(* IEC 61131-3 sources: openplc_school_01/practice04/build/OpenPLC Runtime v3/src, 1 file *)

(* ---- program.st ---- *)
PROGRAM main
  VAR_INPUT
    X0 : BOOL;
    X1 : BOOL;
  END_VAR
  VAR_OUTPUT
    Y0 : BOOL;
  END_VAR

  Y0 := NOT(X1) AND NOT(X0);
END_PROGRAM

CONFIGURATION Config0

  RESOURCE Res0 ON PLC
    TASK task0(INTERVAL := T#20ms,PRIORITY := 1);
    PROGRAM instance0 WITH task0 : main;
  END_RESOURCE
END_CONFIGURATION

(*DBG:char md5[] = "5c376f10d533214feb88b87bce6b503e";*)
(*DBG:/**)
(*DBG: * This file is part of OpenPLC Runtime*)
(*DBG: **)
(*DBG: * Copyright (C) 2023 Autonomy, GP Orcullo*)
(*DBG: * Based on the work by GP Orcullo on Beremiz for uC*)
(*DBG: **)
(*DBG: * This program is free software; you can redistribute it and/or*)
(*DBG: * modify it under the terms of the GNU General Public License*)
(*DBG: * as published by the Free Software Foundation; either version 2*)
(*DBG: * of the License, or (at your option) any later version.*)
(*DBG: **)
(*DBG: * This program is distributed in the hope that it will be useful,*)
(*DBG: * but WITHOUT ANY WARRANTY; without even the implied warranty of*)
(*DBG: * MERCHANTABILITY or FITNESS FOR A PARTICULAR PURPOSE.  See the*)
(*DBG: * GNU General Public License for more details.*)
(*DBG: **)
(*DBG: * You should have received a copy of the GNU General Public License*)
(*DBG: * along with this program; If not, see <http://www.gnu.org/licenses/>.*)
(*DBG: **)
(*DBG: */*)
(*DBG:*)
(*DBG:#include <stdbool.h>*)
(*DBG:*)
(*DBG:#include "iec_types_all.h"*)
(*DBG:#include "POUS.h"*)
(*DBG:*)
(*DBG:#define SAME_ENDIANNESS      0*)
(*DBG:#define REVERSE_ENDIANNESS   1*)
(*DBG:*)
(*DBG:char plc_program_md5[] = "5c376f10d533214feb88b87bce6b503e";*)
(*DBG:*)
(*DBG:uint8_t endianness;*)
(*DBG:*)
(*DBG:*)
(*DBG:extern MAIN RES0__INSTANCE0;*)
(*DBG:*)
(*DBG:static const struct {*)
(*DBG:    void *ptr;*)
(*DBG:    __IEC_types_enum type;*)
(*DBG:} debug_vars[] = {*)
(*DBG:    {&(RES0__INSTANCE0.X0), BOOL_ENUM},*)
(*DBG:    {&(RES0__INSTANCE0.X1), BOOL_ENUM},*)
(*DBG:    {&(RES0__INSTANCE0.Y0), BOOL_ENUM},*)
(*DBG:};*)
(*DBG:*)
(*DBG:#define VAR_COUNT               3*)
(*DBG:*)
(*DBG:uint16_t get_var_count(void)*)
(*DBG:{*)
(*DBG:    return VAR_COUNT;*)
(*DBG:}*)
(*DBG:*)
(*DBG:size_t get_var_size(size_t idx)*)
(*DBG:{*)
(*DBG:    if (idx >= VAR_COUNT)*)
(*DBG:    {*)
(*DBG:        return 0;*)
(*DBG:    }*)
(*DBG:    switch (debug_vars[idx].type) {*)
(*DBG:    case BOOL_ENUM:*)
(*DBG:        return sizeof(BOOL);*)
(*DBG:    default:*)
(*DBG:        return 0;*)
(*DBG:    }*)
(*DBG:}*)
(*DBG:*)
(*DBG:void *get_var_addr(size_t idx)*)
(*DBG:{*)
(*DBG:    void *ptr = debug_vars[idx].ptr;*)
(*DBG:*)
(*DBG:    switch (debug_vars[idx].type) {*)
(*DBG:    case BOOL_ENUM:*)
(*DBG:        return (void *)&((__IEC_BOOL_t *) ptr)->value;*)
(*DBG:    default:*)
(*DBG:        return 0;*)
(*DBG:    }*)
(*DBG:}*)
(*DBG:*)
(*DBG:void force_var(size_t idx, bool forced, void *val)*)
(*DBG:{*)
(*DBG:    void *ptr = debug_vars[idx].ptr;*)
(*DBG:*)
(*DBG:    if (forced) {*)
(*DBG:        size_t var_size = get_var_size(idx);*)
(*DBG:        switch (debug_vars[idx].type) {*)
(*DBG:        case BOOL_ENUM: {*)
(*DBG:            memcpy(&((__IEC_BOOL_t *) ptr)->value, val, var_size);*)
(*DBG:            ((__IEC_BOOL_t *) ptr)->flags |= __IEC_FORCE_FLAG;*)
(*DBG:            break;*)
(*DBG:        }*)
(*DBG:    *)
(*DBG:        default:*)
(*DBG:            break;*)
(*DBG:        }*)
(*DBG:    } else {*)
(*DBG:        switch (debug_vars[idx].type) {*)
(*DBG:        case BOOL_ENUM:*)
(*DBG:            ((__IEC_BOOL_t *) ptr)->flags &= ~__IEC_FORCE_FLAG;*)
(*DBG:            break;*)
(*DBG:        default:*)
(*DBG:            break;*)
(*DBG:        }*)
(*DBG:    }*)
(*DBG:}*)
(*DBG:*)
(*DBG:void swap_bytes(void *ptr, size_t size)*)
(*DBG:{*)
(*DBG:    uint8_t *bytePtr = (uint8_t *)ptr;*)
(*DBG:    size_t i;*)
(*DBG:    for (i = 0; i < size / 2; ++i)*)
(*DBG:    {*)
(*DBG:        uint8_t temp = bytePtr[i];*)
(*DBG:        bytePtr[i] = bytePtr[size - 1 - i];*)
(*DBG:        bytePtr[size - 1 - i] = temp;*)
(*DBG:    }*)
(*DBG:}*)
(*DBG:*)
(*DBG:void trace_reset(void)*)
(*DBG:{*)
(*DBG:    for (size_t i=0; i < VAR_COUNT; i++)*)
(*DBG:    {*)
(*DBG:        force_var(i, false, 0);*)
(*DBG:    }*)
(*DBG:}*)
(*DBG:*)
(*DBG:void set_trace(size_t idx, bool forced, void *val)*)
(*DBG:{*)
(*DBG:    if (idx >= 0 && idx < VAR_COUNT)*)
(*DBG:    {*)
(*DBG:        if (endianness == REVERSE_ENDIANNESS)*)
(*DBG:        {*)
(*DBG:            // Prevent swapping for STRING type*)
(*DBG:            if (debug_vars[idx].type == STRING_ENUM)*)
(*DBG:            {*)
(*DBG:                // Do nothing*)
(*DBG:                ;*)
(*DBG:            }*)
(*DBG:            else*)
(*DBG:            {*)
(*DBG:                swap_bytes(val, get_var_size(idx));*)
(*DBG:            }*)
(*DBG:        }*)
(*DBG:*)
(*DBG:        force_var(idx, forced, val);*)
(*DBG:    }*)
(*DBG:}*)
(*DBG:*)
(*DBG:void set_endianness(uint8_t value)*)
(*DBG:{*)
(*DBG:    if (value == SAME_ENDIANNESS || value == REVERSE_ENDIANNESS)*)
(*DBG:    {*)
(*DBG:        endianness = value;*)
(*DBG:    }*)
(*DBG:}*)
(*DBG:*)
(*FILE:c_blocks.h // Empty file *)
(*FILE:c_blocks.h  *)
(*FILE:c_blocks_code.cpp #include <stdint.h> *)
(*FILE:c_blocks_code.cpp  *)
(*FILE:c_blocks_code.cpp #ifdef ARDUINO *)
(*FILE:c_blocks_code.cpp #include <Arduino.h> *)
(*FILE:c_blocks_code.cpp #endif *)
(*FILE:c_blocks_code.cpp  *)
(*FILE:c_blocks_code.cpp /*********************/ *)
(*FILE:c_blocks_code.cpp /*  IEC Types defs   */ *)
(*FILE:c_blocks_code.cpp /*********************/ *)
(*FILE:c_blocks_code.cpp  *)
(*FILE:c_blocks_code.cpp typedef uint8_t  IEC_BOOL; *)
(*FILE:c_blocks_code.cpp  *)
(*FILE:c_blocks_code.cpp typedef int8_t    IEC_SINT; *)
(*FILE:c_blocks_code.cpp typedef int16_t   IEC_INT; *)
(*FILE:c_blocks_code.cpp typedef int32_t   IEC_DINT; *)
(*FILE:c_blocks_code.cpp typedef int64_t   IEC_LINT; *)
(*FILE:c_blocks_code.cpp  *)
(*FILE:c_blocks_code.cpp typedef uint8_t    IEC_USINT; *)
(*FILE:c_blocks_code.cpp typedef uint16_t   IEC_UINT; *)
(*FILE:c_blocks_code.cpp typedef uint32_t   IEC_UDINT; *)
(*FILE:c_blocks_code.cpp typedef uint64_t   IEC_ULINT; *)
(*FILE:c_blocks_code.cpp  *)
(*FILE:c_blocks_code.cpp typedef uint8_t    IEC_BYTE; *)
(*FILE:c_blocks_code.cpp typedef uint16_t   IEC_WORD; *)
(*FILE:c_blocks_code.cpp typedef uint32_t   IEC_DWORD; *)
(*FILE:c_blocks_code.cpp typedef uint64_t   IEC_LWORD; *)
(*FILE:c_blocks_code.cpp  *)
(*FILE:c_blocks_code.cpp typedef float    IEC_REAL; *)
(*FILE:c_blocks_code.cpp typedef double   IEC_LREAL; *)
(*FILE:c_blocks_code.cpp  *)
(*FILE:c_blocks_code.cpp #ifndef STR_MAX_LEN *)
(*FILE:c_blocks_code.cpp #define STR_MAX_LEN 126 *)
(*FILE:c_blocks_code.cpp #endif *)
(*FILE:c_blocks_code.cpp  *)
(*FILE:c_blocks_code.cpp #ifndef STR_LEN_TYPE *)
(*FILE:c_blocks_code.cpp #define STR_LEN_TYPE int8_t *)
(*FILE:c_blocks_code.cpp #endif *)
(*FILE:c_blocks_code.cpp  *)
(*FILE:c_blocks_code.cpp typedef STR_LEN_TYPE __strlen_t; *)
(*FILE:c_blocks_code.cpp typedef struct { *)
(*FILE:c_blocks_code.cpp     __strlen_t len; *)
(*FILE:c_blocks_code.cpp     uint8_t body[STR_MAX_LEN]; *)
(*FILE:c_blocks_code.cpp } IEC_STRING; *)
(*FILE:c_blocks_code.cpp  *)
